(* PLC project traffic_lights, Beremiz Unnamed 1 *)
(* stored: creationDateTime 2012-09-04T16:16:33, modificationDateTime 2023-04-04T09:09:43 *)

FUNCTION_BLOCK traffic_light_sequence
  VAR_INPUT
    SWITCH_BUTTON : BOOL;
    PEDESTRIAN_BUTTON : BOOL;
  END_VAR
  VAR_OUTPUT
    RED_LIGHT : BOOL;
    ORANGE_LIGHT : BOOL;
    GREEN_LIGHT : BOOL;
    PEDESTRIAN_RED_LIGHT : BOOL;
    PEDESTRIAN_GREEN_LIGHT : BOOL;
  END_VAR
  VAR
    TON1 : TON;
    TON2 : TON;
    ALLOW_CARS : BOOL;
    WARN_CARS : BOOL;
    STOP_CARS : BOOL;
    ALLOW_PEDESTRIANS : BOOL;
    STOP_PEDESTRIANS : BOOL;
    TON3 : TON;
    R_TRIG0 : R_TRIG;
    R_TRIG1 : R_TRIG;
    SR0 : SR;
  END_VAR
  VAR  (* added by the conversion: wires and edge detectors of the diagram *)
    _OR35_OUT : BOOL;
  END_VAR

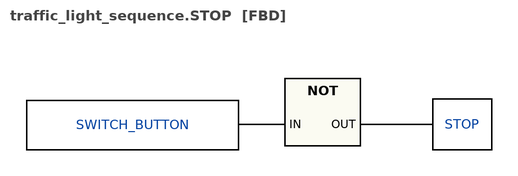
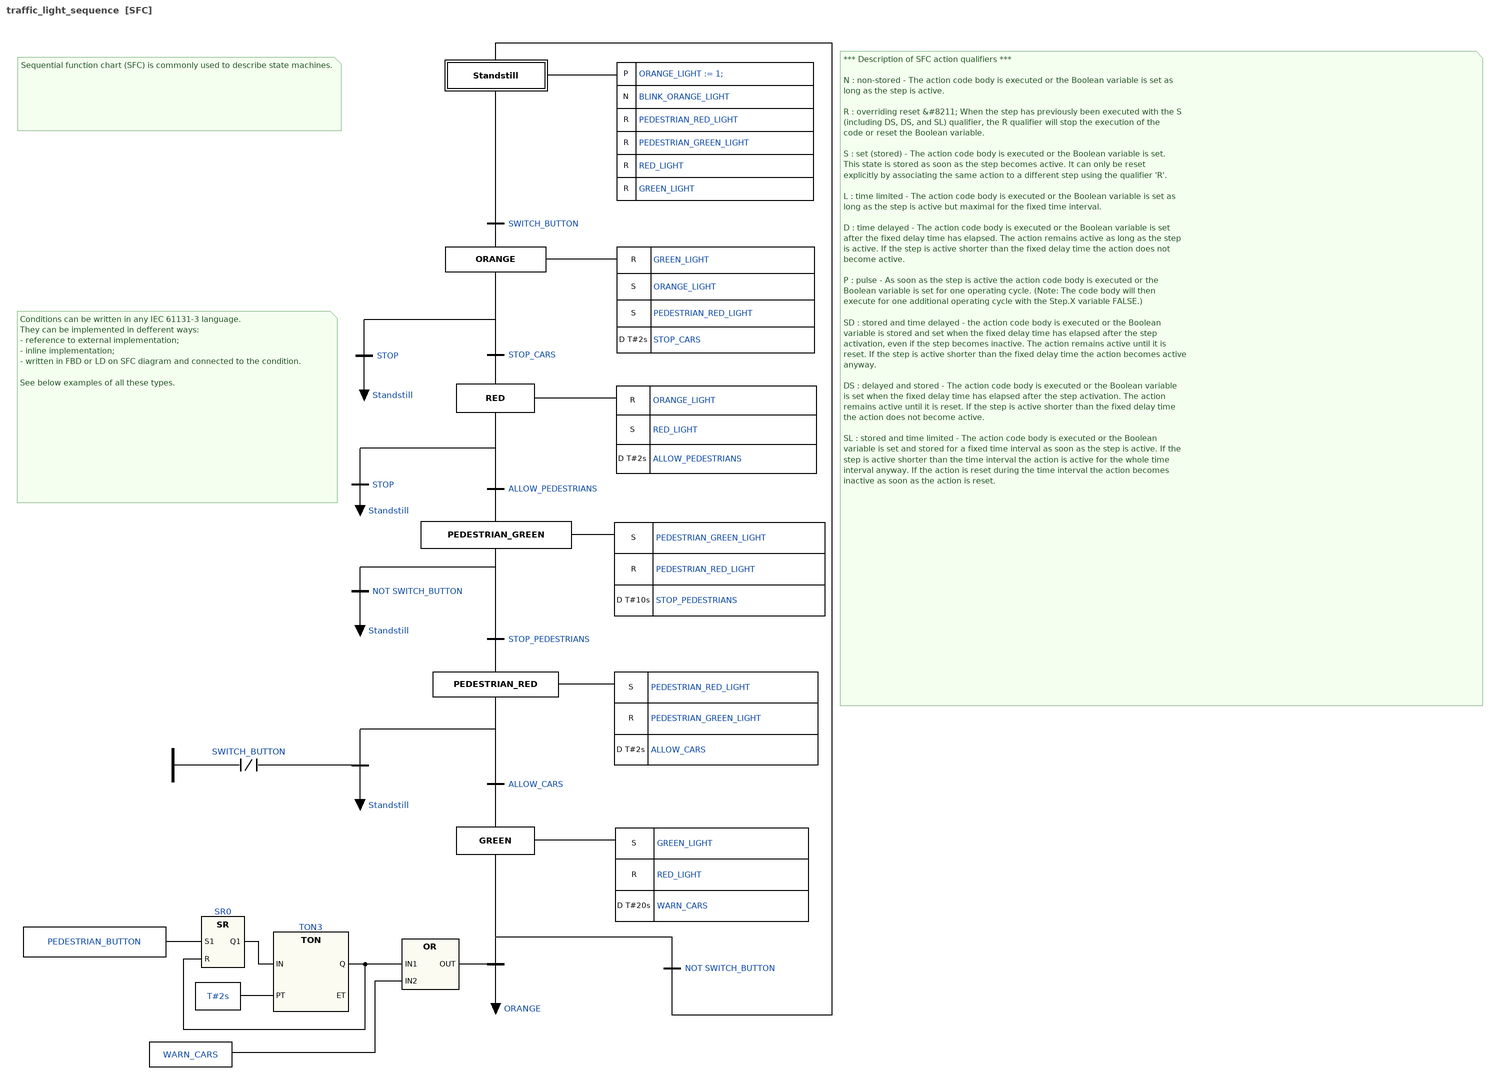
(* *** Description of SFC action qualifiers ***

N : non-stored - The action code body is executed or the Boolean variable is set as
long as the step is active.

R : overriding reset &#8211; When the step has previously been executed with the S
(including DS, DS, and SL) qualifier, the R qualifier will stop the execution of the
code or reset the Boolean variable.

S : set (stored) - The action code body is executed or the Boolean variable is set.
This state is stored as soon as the step becomes active. It can only be reset
explicitly by associating the same action to a different step using the qualifier 'R'.

L : time limited - The action code body is executed or the Boolean variable is set as
long as the step is active but maximal for the fixed time interval.

D : time delayed - The action code body is executed or the Boolean variable is set
after the fixed delay time has elapsed. The action remains active as long as the step
is active. If the step is active shorter than the fixed delay time the action does not
become active.

P : pulse - As soon as the step is active the action code body is executed or the
Boolean variable is set for one operating cycle. (Note: The code body will then
execute for one additional operating cycle with the Step.X variable FALSE.)

SD : stored and time delayed - the action code body is executed or the Boolean
variable is stored and set when the fixed delay time has elapsed after the step
activation, even if the step becomes inactive. The action remains active until it is
reset. If the step is active shorter than the fixed delay time the action becomes active
anyway.

DS : delayed and stored - The action code body is executed or the Boolean variable
is set when the fixed delay time has elapsed after the step activation. The action
remains active until it is reset. If the step is active shorter than the fixed delay time
the action does not become active.

SL : stored and time limited - The action code body is executed or the Boolean
variable is set and stored for a fixed time interval as soon as the step is active. If the
step is active shorter than the time interval the action is active for the whole time
interval anyway. If the action is reset during the time interval the action becomes
inactive as soon as the action is reset. *)
(* Conditions can be written in any IEC 61131-3 language.
They can be implemented in defferent ways:
- reference to external implementation;
- inline implementation;
- written in FBD or LD on SFC diagram and connected to the condition.

See below examples of all these types. *)
(* Sequential function chart (SFC) is commonly used to describe state machines. *)
INITIAL_STEP Standstill:
  STANDSTILL_INLINE1(P);
  BLINK_ORANGE_LIGHT(N);
  PEDESTRIAN_RED_LIGHT(R);
  PEDESTRIAN_GREEN_LIGHT(R);
  RED_LIGHT(R);
  GREEN_LIGHT(R);
  COMPUTE_FUNCTION_BLOCKS(S);
END_STEP
ACTION STANDSTILL_INLINE1:
  ORANGE_LIGHT := 1;
END_ACTION
TRANSITION FROM Standstill TO ORANGE
  := SWITCH_BUTTON;
END_TRANSITION
STEP ORANGE:
  GREEN_LIGHT(R);
  ORANGE_LIGHT(S);
  PEDESTRIAN_RED_LIGHT(S);
  STOP_CARS(D, T#2s);
END_STEP
TRANSITION FROM ORANGE TO RED
  := STOP_CARS;
END_TRANSITION
TRANSITION FROM ORANGE TO Standstill  (* STOP *)
  := NOT SWITCH_BUTTON;
END_TRANSITION
STEP RED:
  ORANGE_LIGHT(R);
  RED_LIGHT(S);
  ALLOW_PEDESTRIANS(D, T#2s);
END_STEP
TRANSITION FROM RED TO PEDESTRIAN_GREEN
  := ALLOW_PEDESTRIANS;
END_TRANSITION
TRANSITION FROM RED TO Standstill  (* STOP *)
  := NOT SWITCH_BUTTON;
END_TRANSITION
STEP PEDESTRIAN_GREEN:
  PEDESTRIAN_GREEN_LIGHT(S);
  PEDESTRIAN_RED_LIGHT(R);
  STOP_PEDESTRIANS(D, T#10s);
END_STEP
TRANSITION FROM PEDESTRIAN_GREEN TO Standstill
  := NOT SWITCH_BUTTON;
END_TRANSITION
TRANSITION FROM PEDESTRIAN_GREEN TO PEDESTRIAN_RED
  := STOP_PEDESTRIANS;
END_TRANSITION
STEP PEDESTRIAN_RED:
  PEDESTRIAN_RED_LIGHT(S);
  PEDESTRIAN_GREEN_LIGHT(R);
  ALLOW_CARS(D, T#2s);
END_STEP
TRANSITION FROM PEDESTRIAN_RED TO Standstill
  := NOT SWITCH_BUTTON;
END_TRANSITION
TRANSITION FROM PEDESTRIAN_RED TO GREEN
  := ALLOW_CARS;
END_TRANSITION
STEP GREEN:
  GREEN_LIGHT(S);
  RED_LIGHT(R);
  WARN_CARS(D, T#20s);
END_STEP
TRANSITION FROM GREEN TO ORANGE
  := _OR35_OUT;
END_TRANSITION
TRANSITION FROM GREEN TO Standstill
  := NOT SWITCH_BUTTON;
END_TRANSITION
ACTION COMPUTE_FUNCTION_BLOCKS:  (* blocks drawn on the SFC sheet *)
  SR0(S1 := PEDESTRIAN_BUTTON, R := TON3.Q);
  TON3(IN := SR0.Q1, PT := T#2s);
  _OR35_OUT := TON3.Q OR WARN_CARS;
END_ACTION

ACTION BLINK_ORANGE_LIGHT:
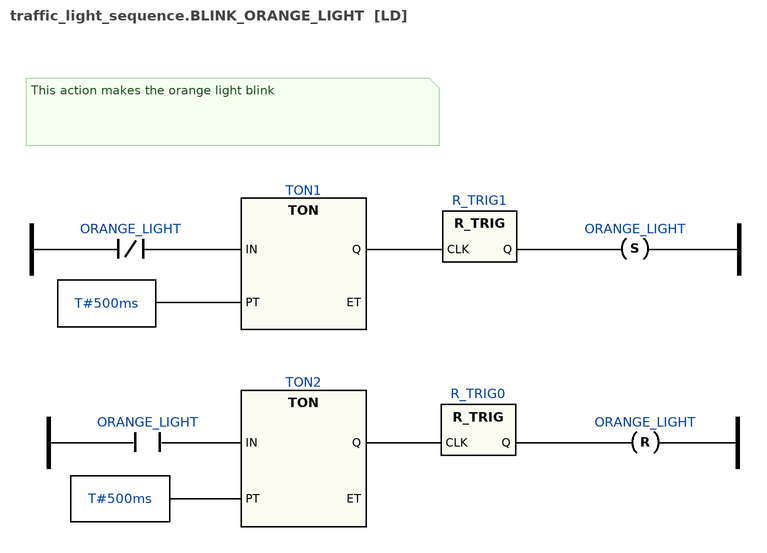
(* LD diagram, written out as Structured Text *)
(* This action makes the orange light blink *)
TON1(IN := NOT ORANGE_LIGHT, PT := T#500ms);
R_TRIG1(CLK := TON1.Q);
IF R_TRIG1.Q THEN ORANGE_LIGHT := TRUE; END_IF;
TON2(IN := ORANGE_LIGHT, PT := T#500ms);
R_TRIG0(CLK := TON2.Q);
IF R_TRIG0.Q THEN ORANGE_LIGHT := FALSE; END_IF;
END_ACTION
END_FUNCTION_BLOCK

PROGRAM main_program
  VAR
    SwitchButton AT %IX0.0.0 : BOOL;
    PedestrianButton AT %IX0.0.1 : BOOL;
    RedLight AT %QX0.0.0 : BOOL;
    OrangeLight AT %QX0.0.1 : BOOL;
    GreenLight AT %QX0.0.2 : BOOL;
    PedestrianRedLight AT %QX0.0.3 : BOOL;
    PedestrianGreenLight AT %QX0.0.4 : BOOL;
  END_VAR
  VAR
    traffic_light_sequence0 : traffic_light_sequence;
  END_VAR

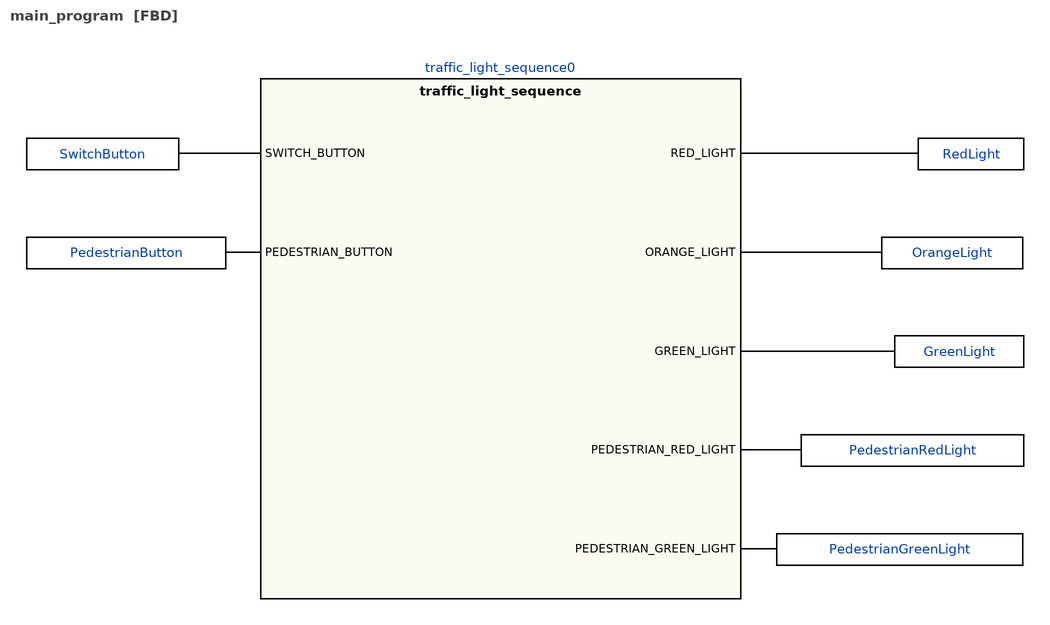
(* FBD diagram, written out as Structured Text *)
traffic_light_sequence0(SWITCH_BUTTON := SwitchButton, PEDESTRIAN_BUTTON := PedestrianButton);
RedLight := traffic_light_sequence0.RED_LIGHT;
OrangeLight := traffic_light_sequence0.ORANGE_LIGHT;
GreenLight := traffic_light_sequence0.GREEN_LIGHT;
PedestrianRedLight := traffic_light_sequence0.PEDESTRIAN_RED_LIGHT;
PedestrianGreenLight := traffic_light_sequence0.PEDESTRIAN_GREEN_LIGHT;
END_PROGRAM

CONFIGURATION config
  RESOURCE resource1 ON PLC
    TASK test_task(INTERVAL := T#500ms, PRIORITY := 0);
    PROGRAM main_instance WITH test_task : main_program;
  END_RESOURCE
END_CONFIGURATION
